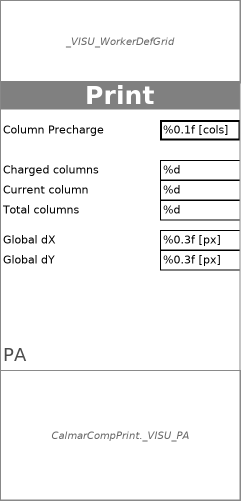
VISUALIZATION _VISU_WorkerDefGrid_Print  // 241x501
VAR_IN_OUT
  m_Inst : FB_WorkerDefGrid_Print;
END_VAR
    Frame (0,0 241x83)
        shows _VISU_WorkerDefGrid(m_Inst := m_Inst)
    Rectangle (0,120 160x20), "Column Precharge"
    Rectangle (160,120 80x20), "%0.1f [cols]", text variable: m_Inst._fColumnsToPrecharge
        OnMouseDown: write the text variable via Default
    Label (0,340 240x30), "PA"
    Rectangle (0,80 240x30), "Print", colour toggle: m_Inst._pAttachedCt <> 0
    Rectangle (0,160 160x20), "Charged columns"
    Rectangle (160,160 80x20), "%d", text variable: m_Inst.nChargedColumns
    Rectangle (0,180 160x20), "Current column", tooltip "Current columen relative to Worker Attach"
    Rectangle (160,180 80x20), "%d", text variable: m_Inst.fCurrentColumnPos
    Rectangle (0,200 160x20), "Total columns"
    Rectangle (160,200 80x20), "%d", text variable: m_Inst.sDefGridSettings.nGridSizeX
    Frame (0,370 241x131)
        shows CalmarCompPrint._VISU_PA(m_Inst := m_Inst.fbPa)
    Rectangle (0,230 160x20), "Global dX"
    Rectangle (160,230 80x20), "%0.3f [px]", text variable: m_Inst._fDxGlobalShift
    Rectangle (0,250 160x20), "Global dY"
    Rectangle (160,250 80x20), "%0.3f [px]", text variable: m_Inst._fDyGlobalShift
END_VISUALIZATION

(* stored: Version 1.1.0.1, ProductVersion 3.1.4024.3
   Visu _VISU_WorkerDefGrid_Print: Id {637c3541-8029-4103-a7ba-3d7ba899339f} *)
